TYPE AnalogController :
STRUCT
	pv : REAL;
	cv : REAL;
	tv : REAL;
	maxValue : REAL;
	cvController : FB_ControlRampGenerator;
END_STRUCT
END_TYPE

(* stored: Version 1.1.0.1, ProductVersion 3.1.4026.11
   DUT AnalogController: Id {4bd54bf5-cb89-4b47-8a5b-7834b54c8812} *)
